// TIA Portal V18 export
FUNCTION_BLOCK "Hauptablauf"   // FB1000, LAD
TITLE = Hauptablauf
{ S7_Optimized_Access := 'FALSE' }
// stored: SetENOAutomatically false
   VAR_TEMP
      MIdx : Int;
   END_VAR
BEGIN

REGION Network 1 (SCL)
   "DB_BA".bSKZähler := 0;
END_REGION

REGION Network 2
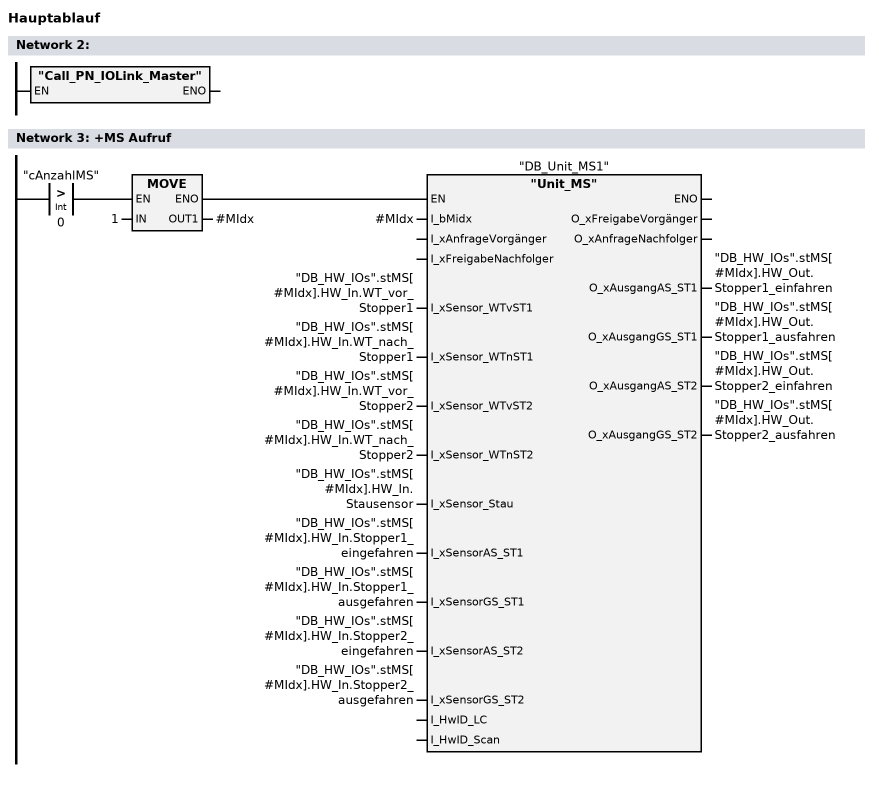
   RUNG wire#powerrail
      "Call_PN_IOLink_Master"()
   END_RUNG
   // the same network as SCL:
   "Call_PN_IOLink_Master"();
END_REGION

REGION Network 3: +MS Aufruf
   RUNG wire#powerrail
      { S7_Templates := "SrcType := Int" } GT_Contact(in1 := "cAnzahlMS", in2 := 0)
      Move(in := 1, out1 => #MIdx)
      "DB_Unit_MS1"(I_bMidx := #MIdx, I_xAnfrageVorgänger :=, I_xFreigabeNachfolger :=, I_xSensor_WTvST1 := "DB_HW_IOs".stMS[#MIdx].HW_In.WT_vor_Stopper1, I_xSensor_WTnST1 := "DB_HW_IOs".stMS[#MIdx].HW_In.WT_nach_Stopper1, I_xSensor_WTvST2 := "DB_HW_IOs".stMS[#MIdx].HW_In.WT_vor_Stopper2, I_xSensor_WTnST2 := "DB_HW_IOs".stMS[#MIdx].HW_In.WT_nach_Stopper2, I_xSensor_Stau := "DB_HW_IOs".stMS[#MIdx].HW_In.Stausensor, I_xSensorAS_ST1 := "DB_HW_IOs".stMS[#MIdx].HW_In.Stopper1_eingefahren, I_xSensorGS_ST1 := "DB_HW_IOs".stMS[#MIdx].HW_In.Stopper1_ausgefahren, I_xSensorAS_ST2 := "DB_HW_IOs".stMS[#MIdx].HW_In.Stopper2_eingefahren, I_xSensorGS_ST2 := "DB_HW_IOs".stMS[#MIdx].HW_In.Stopper2_ausgefahren, I_HwID_LC :=, I_HwID_Scan :=, O_xFreigabeVorgänger =>, O_xAnfrageNachfolger =>, O_xAusgangAS_ST1 => "DB_HW_IOs".stMS[#MIdx].HW_Out.Stopper1_einfahren, O_xAusgangGS_ST1 => "DB_HW_IOs".stMS[#MIdx].HW_Out.Stopper1_ausfahren, O_xAusgangAS_ST2 => "DB_HW_IOs".stMS[#MIdx].HW_Out.Stopper2_einfahren, O_xAusgangGS_ST2 => "DB_HW_IOs".stMS[#MIdx].HW_Out.Stopper2_ausfahren)
   END_RUNG
   // the same network as SCL:
   IF "cAnzahlMS" > 0 THEN
       #MIdx := 1;
       "DB_Unit_MS1"(I_bMidx := #MIdx,   // "Unit_MS"
                     I_xSensor_WTvST1 := "DB_HW_IOs".stMS[#MIdx].HW_In.WT_vor_Stopper1,
                     I_xSensor_WTnST1 := "DB_HW_IOs".stMS[#MIdx].HW_In.WT_nach_Stopper1,
                     I_xSensor_WTvST2 := "DB_HW_IOs".stMS[#MIdx].HW_In.WT_vor_Stopper2,
                     I_xSensor_WTnST2 := "DB_HW_IOs".stMS[#MIdx].HW_In.WT_nach_Stopper2,
                     I_xSensor_Stau := "DB_HW_IOs".stMS[#MIdx].HW_In.Stausensor,
                     I_xSensorAS_ST1 := "DB_HW_IOs".stMS[#MIdx].HW_In.Stopper1_eingefahren,
                     I_xSensorGS_ST1 := "DB_HW_IOs".stMS[#MIdx].HW_In.Stopper1_ausgefahren,
                     I_xSensorAS_ST2 := "DB_HW_IOs".stMS[#MIdx].HW_In.Stopper2_eingefahren,
                     I_xSensorGS_ST2 := "DB_HW_IOs".stMS[#MIdx].HW_In.Stopper2_ausgefahren,
                     O_xAusgangAS_ST1 => "DB_HW_IOs".stMS[#MIdx].HW_Out.Stopper1_einfahren,
                     O_xAusgangGS_ST1 => "DB_HW_IOs".stMS[#MIdx].HW_Out.Stopper1_ausfahren,
                     O_xAusgangAS_ST2 => "DB_HW_IOs".stMS[#MIdx].HW_Out.Stopper2_einfahren,
                     O_xAusgangGS_ST2 => "DB_HW_IOs".stMS[#MIdx].HW_Out.Stopper2_ausfahren);
   END_IF;
END_REGION
END_FUNCTION_BLOCK
